{attribute 'qualified_only'}
{attribute 'to_string'}
{attribute 'strict'}
TYPE E_DATA_CTRL :
(
  NULL,
	INIT  := 10,
  READ  := 20,
  WRITE := 30
)UINT;
END_TYPE

(* stored: Version 1.1.0.1, ProductVersion 3.1.4026.20
   DUT E_DATA_CTRL: Id {1c91b981-307e-4de1-b9a2-a68010cb78cd} *)
